ABB RobotStudio station: Compas_RRC_Course.rspag

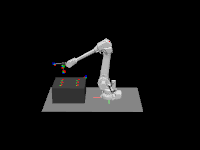
--- station ---
Station Compas_RRC_Course (saved by RobotStudio 20.4.9280.0)
Controller vIRB4600-40-255_RRC
  mechanical unit ROB_1: IRB4600_40_255_C_01, 6 joints, base frame (0, 0, 0) mm
Layout (positions relative to the parent item):
  - IRB4600_40_255_C_01 [mechanism] at (0, 0, 0) mm; joint values [0, -0.1281, 0.6287, 3.1416, 0.5005, 3.1416] (rad or m)
      links: Base, Link1, Link2, Link3, Link4, Link5, Link6
  - Table [part]
  - Ground [part]
  - Tool [graphiccomponentgroup] at (1368.26, 0, 1125.08) mm, rotated rx -13.36 ry 90 rz -13.36 deg
    - Tool X TubeTrace [smart component] at (0, 0, 0) mm
        properties: TraceObject=(none); ActiveTube=(none); Mechanism=IRB4600_40_255_C_01; Flange=Tool0; Parent=(none); Flange Offset=[0.26 0 0.06]; Tube Diameter=0.03; Color (RGB)=[255 255 255]; Color=-65536; Min Distance=0.001; Redraw Rate (ms)=10; NoOfBodies=210; Remove Geometry=true; Transient=false
        signals: DI Execute, DI NewTrace, DI Clear, DO TraceCreated
    - Tool Y TubeTrace [smart component] at (0, 0, 0) mm
        properties: TraceObject=(none); ActiveTube=(none); Mechanism=IRB4600_40_255_C_01; Flange=Tool0; Parent=(none); Flange Offset=[0 0.26 0.06]; Tube Diameter=0.03; Color (RGB)=[255 255 255]; Color=-16711872; Min Distance=0.001; Redraw Rate (ms)=10; NoOfBodies=208; Remove Geometry=true; Transient=false
        signals: DI Execute, DI NewTrace, DI Clear, DO TraceCreated
    - Tool Z TubeTrace [smart component] at (0, 0, 0) mm
        properties: TraceObject=(none); ActiveTube=(none); Mechanism=IRB4600_40_255_C_01; Flange=Tool0; Parent=(none); Flange Offset=[0 0 0.32]; Tube Diameter=0.03; Color (RGB)=[255 255 255]; Color=-16776961; Min Distance=0.001; Redraw Rate (ms)=10; NoOfBodies=210; Remove Geometry=true; Transient=false
        signals: DI Execute, DI NewTrace, DI Clear, DO TraceCreated
    - Tool X [part] at (0, 0, 0) mm
    - Tool Y [part] at (0, 0, 0) mm
    - Tool Z [part] at (0, 0, 0) mm
    - Base [part] at (1428.26, 0, 1185.08) mm, rotated rx 180 ry 0 rz -180 deg
Attachment: Tool is attached to IRB4600_40_255_C_01 / Link6
Station logic (signal -> signal, property => property):
  vIRB4600-40-255_RRC.doPrintTX -> Tool X TubeTrace.Execute
  vIRB4600-40-255_RRC.doPrintTY -> Tool Y TubeTrace.Execute
  vIRB4600-40-255_RRC.doPrintTZ -> Tool Z TubeTrace.Execute
Targets, tools, work objects and paths stored in the station and not in the controller backup, written as RAPID:
! task T_ROB1
MODULE X000_Tests
  PROC r_X000_Parh_Z()
    MoveJ pZStart,v200,fine,t_X000_Tool_Z\WObj:=ob_X000_Workplace;
    MoveL pZ1,v200,fine,t_X000_Tool_Z\WObj:=ob_X000_Workplace;
    MoveL pZ2,v200,fine,t_X000_Tool_Z\WObj:=ob_X000_Workplace;
  ENDPROC
  PROC r_X000_Parh_X()
    MoveJ pXStart,v200,fine,t_X000_Tool_X\WObj:=ob_X000_Workplace;
    MoveL pX1,v200,fine,t_X000_Tool_X\WObj:=ob_X000_Workplace;
    MoveL pX2,v200,fine,t_X000_Tool_X\WObj:=ob_X000_Workplace;
  ENDPROC
  PROC r_X000_Parh_Y()
    MoveJ pYStart,v200,fine,t_X000_Tool_Y\WObj:=ob_X000_Workplace;
    MoveL pY1,v200,fine,t_X000_Tool_Y\WObj:=ob_X000_Workplace;
    MoveL pY2,v200,fine,t_X000_Tool_Y\WObj:=ob_X000_Workplace;
  ENDPROC
ENDMODULE


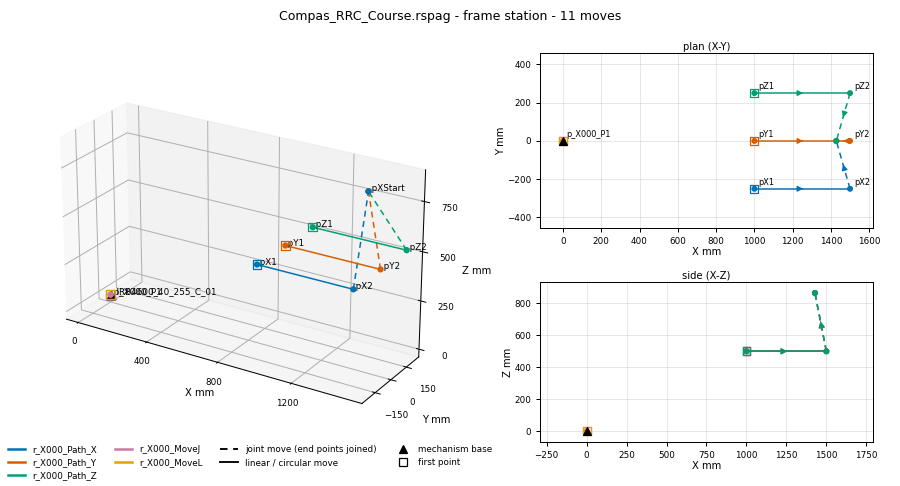
[picture p0: tool path of Compas_RRC_Course.rspag in frame station, 11 of 14 moves have a stored position in this frame; points joined in program order, loops and branches not executed]
--- Backups/vIRB4600-40-255_RRC/RAPID/TASK1/PROGMOD/X000_DataTask_1.mod ---
MODULE X000_DataTask_1
    !***********************************************************************************
    !
    ! ETH Zurich / NCCR Digital Fabrication
    ! HIB C51 / Stefano-Franscini-Platz 1
    ! CH-8093 Zürich
    !
    !***********************************************************************************
    !
    ! PROJECT     :  X000 Default
    !
    ! FUNCTION    :  Includ all Task Data's for Project
    !
    ! AUTHOR      :  Philippe Fleischmann
    !
    ! EMAIL       :  fleischmann@arch.ethz.ch
    !
    ! HISTORY     :  2019.12.04
    !
    ! Copyright   :  ETH Zürich (CH) 2019
    !
    !***********************************************************************************

    !************************************************
    ! Declaration :     bool
    !************************************************
    !

    !************************************************
    ! Declaration :     num
    !************************************************
    !

    !************************************************
    ! Declaration :     string
    !************************************************
    !

    !************************************************
    ! Declaration :     tooldata
    !************************************************
    !
    TASK PERS tooldata t_X000_Tool:=[TRUE,[[0,0,0],[1,0,0,0]],[1,[0,0,0],[1,0,0,0],0.1,0.1,0.1]];
    !
    TASK PERS tooldata t_X000_Tool_X:=[TRUE,[[260,0,60],[0.707106781,0,0.707106781,0]],[15,[0,0,60],[1,0,0,0],0.1,0.1,0.1]];
    TASK PERS tooldata t_X000_Tool_Y:=[TRUE,[[0,260,60],[0.707106781,-0.707106781,0,0]],[15,[0,0,60],[1,0,0,0],0.1,0.1,0.1]];
    TASK PERS tooldata t_X000_Tool_Z:=[TRUE,[[0,0,320],[1,0,0,0]],[15,[0,0,60],[1,0,0,0],0.1,0.1,0.1]];

    !************************************************
    ! Declaration :     wobjdata
    !************************************************
    !
    TASK PERS wobjdata ob_X000_Wobjdata:=[FALSE,TRUE,"",[[0,0,0],[1,0,0,0]],[[0,0,0],[1,0,0,0]]];
    !
    TASK PERS wobjdata ob_X000_Workplace:=[FALSE,TRUE,"",[[750,-500,500],[1,0,0,0]],[[0,0,0],[1,0,0,0]]];

    !************************************************
    ! Declaration :     jointtarget
    !************************************************
    !
    TASK PERS jointtarget jp_X000_Jointtarget:=[[0,0,0,0,0,0],[9E9,9E9,9E9,9E9,9E9,9E9]];
    !
    TASK PERS jointtarget jp_X000_Start:=[[1.2417E-18,-7.34132,36.0203,180,28.679,180],[9E+9,9E+9,9E+9,9E+9,9E+9,9E+9]];

    !************************************************
    ! Declaration :     robtarget
    !************************************************
    !
    TASK PERS robtarget p_X000_Robtarget:=[[0,0,0],[1,0,0,0],[0,0,0,0],[9E9,9E9,9E9,9E9,9E9,9E9]];

	CONST robtarget pXStart:=[[678.26315348,500,365.080626614],[0,0,1,0],[0,2,2,0],[9E+09,9E+09,9E+09,9E+09,9E+09,9E+09]];
	CONST robtarget pX1:=[[250.000037817,249.999985042,-0.000049799],[-0.000000001,0,1,-0.000000028],[-1,1,2,0],[9E+09,9E+09,9E+09,9E+09,9E+09,9E+09]];
	CONST robtarget pX2:=[[750.000017046,249.999996608,-0.000043508],[-0.000000001,-0.000000024,1,0],[-1,1,2,0],[9E+09,9E+09,9E+09,9E+09,9E+09,9E+09]];

    CONST robtarget pYStart:=[[678.26315348,500,365.080626614],[0,0,1,0],[0,-1,0,0],[9E+09,9E+09,9E+09,9E+09,9E+09,9E+09]];
	CONST robtarget pY1:=[[250.000037817,499.999985042,-0.000049799],[-0.000000001,0,1,-0.000000028],[0,-1,0,0],[9E+09,9E+09,9E+09,9E+09,9E+09,9E+09]];
	CONST robtarget pY2:=[[750.000017046,499.999996608,-0.000043508],[-0.000000001,-0.000000024,1,0],[0,-1,0,0],[9E+09,9E+09,9E+09,9E+09,9E+09,9E+09]];

    CONST robtarget pZStart:=[[678.26315348,500,365.080626614],[0,0,1,0],[0,0,0,0],[9E+09,9E+09,9E+09,9E+09,9E+09,9E+09]];
	CONST robtarget pZ1:=[[250.000037817,749.999985042,-0.000077799],[-0.000000001,0,1,-0.000000028],[0,-1,0,0],[9E+09,9E+09,9E+09,9E+09,9E+09,9E+09]];
	CONST robtarget pZ2:=[[750.000017046,749.999996608,-0.000071508],[-0.000000001,-0.000000024,1,0],[0,0,0,0],[9E+09,9E+09,9E+09,9E+09,9E+09,9E+09]];

    !************************************************
    ! Declaration :     speeddata
    !************************************************
    !
    TASK PERS speeddata v_X000_Speed:=[0,0,0,0];

ENDMODULE

--- Backups/vIRB4600-40-255_RRC/RAPID/TASK1/PROGMOD/X000_Demo.mod ---
MODULE X000_Demo
    !***********************************************************************************
    !
    ! ETH Zürich / Robotic Fabrication Lab
    ! HIB C 13 / Stefano-Franscini-Platz 1
    ! CH-8093 Zürich
    !
    !***********************************************************************************
    !
    ! PROJECT     :  X000_Default
    !
    ! FUNCTION    :  Demo
    !
    ! AUTHOR      :  Philippe Fleischmann
    !
    ! EMAIL       :  fleischmann@arch.ethz.ch
    !
    ! HISTORY     :  2021.01.14
    !
    ! Copyright   :  ETH Zürich (CH) 2021
    !
    !***********************************************************************************

    !************************************************
    ! Function    :     Demo x y and z path
    ! Programmer  :     Philippe Fleischmann
    ! Date        :     2021.01.14
    !***************** ETH Zürich *******************
    !
    PROC main()
        !
        ! Move to start point
        MoveAbsJ jp_X000_Start,v200,fine,tool0;
        !
        ! Test paths
        r_X000_Path_X;
        r_X000_Path_Y;
        r_X000_Path_Z;
        !
        ! Move to start point
        MoveAbsJ jp_X000_Start,v200,fine,tool0;
        !
        RETURN ;
    ERROR
        ! Placeholder for Error Code...
    ENDPROC

    !************************************************
    ! Function    :     Print Path red
    ! Programmer  :     Philippe Fleischmann
    ! Date        :     2021.01.14
    !***************** ETH Zürich *******************
    !
    PROC r_X000_Path_X()
        !
        ! Move to print start
        MoveJ pX1,v200,fine,t_X000_Tool_X\WObj:=ob_X000_Workplace;
        !
        ! Start print
        SetDO doPrintTX,1;
        !
        ! Print
        MoveL pX2,v200,fine,t_X000_Tool_X\WObj:=ob_X000_Workplace;
        !
        ! Stop pring
        SetDO doPrintTX,0;
        !
        ! Move back to start point
        MoveJ pXStart,v200,fine,t_X000_Tool_X\WObj:=ob_X000_Workplace;
        !
        RETURN ;
    ERROR
        ! Placeholder for Error Code...
    ENDPROC

    !************************************************
    ! Function    :     Print Path green
    ! Programmer  :     Philippe Fleischmann
    ! Date        :     2021.01.14
    !***************** ETH Zürich *******************
    !
    PROC r_X000_Path_Y()
        !
        ! Move to print start
        MoveJ pY1,v200,fine,t_X000_Tool_Y\WObj:=ob_X000_Workplace;
        !
        ! Start print
        SetDO doPrintTY,1;
        !
        ! Print
        MoveL pY2,v200,fine,t_X000_Tool_Y\WObj:=ob_X000_Workplace;
        !
        ! Stop pring
        SetDO doPrintTY,0;
        !
        ! Move back to start point
        MoveJ pYStart,v200,fine,t_X000_Tool_Y\WObj:=ob_X000_Workplace;
        !
        RETURN ;
    ERROR
        ! Placeholder for Error Code...
    ENDPROC

    !************************************************
    ! Function    :     Print Path blue
    ! Programmer  :     Philippe Fleischmann
    ! Date        :     2021.01.14
    !***************** ETH Zürich *******************
    !
    PROC r_X000_Path_Z()
        !
        ! Move to print start
        MoveJ pZ1,v200,fine,t_X000_Tool_Z\WObj:=ob_X000_Workplace;
        !
        ! Start print
        SetDO doPrintTZ,1;
        !
        ! Print
        MoveL pZ2,v200,fine,t_X000_Tool_Z\WObj:=ob_X000_Workplace;
        !
        ! Stop pring
        SetDO doPrintTZ,0;
        !
        ! Move back to start point
        MoveJ pZStart,v200,fine,t_X000_Tool_Z\WObj:=ob_X000_Workplace;
        !
        RETURN ;
    ERROR
        ! Placeholder for Error Code...
    ENDPROC

ENDMODULE

--- Backups/vIRB4600-40-255_RRC/RAPID/TASK1/PROGMOD/X000_Motion.mod ---
MODULE X000_Motion
    !***********************************************************************************
    !
    ! ETH Zürich / Robotic Fabrication Lab
    ! HIB C 13 / Stefano-Franscini-Platz 1
    ! CH-8093 Zürich
    !
    !***********************************************************************************
    !
    ! PROJECT     :  X000_Default
    !
    ! FUNCTION    :  Motion Types
    !
    ! AUTHOR      :  Philippe Fleischmann
    !
    ! EMAIL       :  fleischmann@arch.ethz.ch
    !
    ! HISTORY     :  2020.01.09
    !
    ! Copyright   :  ETH Zürich (CH) 2017
    !
    !***********************************************************************************

    !************************************************
    ! Declaration :     jointtarget
    !************************************************
    !
    TASK PERS jointtarget jp_X000_P1:=[[0,0,0,0,0,0],[9E9,9E9,9E9,9E9,9E9,9E9]];

    !************************************************
    ! Declaration :     robtarget
    !************************************************
    !
    TASK PERS robtarget p_X000_P1:=[[0,0,0],[1,0,0,0],[0,0,0,0],[9E9,9E9,9E9,9E9,9E9,9E9]];

    !************************************************
    ! Function    :     Move absolute Joint
    ! Programmer  :     Philippe Fleischmann
    ! Date        :     2020.01.07
    !***************** ETH Zürich *******************
    !
    PROC r_X000_MoveAbsJ()
        !
        ! MoveAbsJ
        MoveAbsJ jp_X000_P1,v100,fine,tool0;
        !
        RETURN ;
    ERROR
        ! Placeholder for Error Code...
    ENDPROC

    !************************************************
    ! Function    :     Move Joint
    ! Programmer  :     Philippe Fleischmann
    ! Date        :     2020.01.07
    !***************** ETH Zürich *******************
    !
    PROC r_X000_MoveJ()
        !
        ! MoveJ
        MoveJ p_X000_P1,v100,fine,tool0\WObj:=wobj0;
        !
        RETURN ;
    ERROR
        ! Placeholder for Error Code...
    ENDPROC

    !************************************************
    ! Function    :     Move Linear
    ! Programmer  :     Philippe Fleischmann
    ! Date        :     2020.01.07
    !***************** ETH Zürich *******************
    !
    PROC r_X000_MoveL()
        !
        ! MoveL
        MoveL p_X000_P1,v100,fine,tool0\WObj:=wobj0;
        !
        RETURN ;
    ERROR
        ! Placeholder for Error Code...
    ENDPROC

ENDMODULE

--- Backups/vIRB4600-40-255_RRC/SYSPAR/EIO.cfg ---
EIO:CFG_1.0:6:1::
#
INDUSTRIAL_NETWORK:

      -Name "PROFINET" -Connection "PROFINET Network"\
      -Label "PROFINET Controller/Device Network" -StationName ""
#
EIO_CROSS:

      -Name "FP1" -Res "diMaFP1" -Act1 "doMaFP1"

      -Name "FP2" -Res "diMaFP2" -Act1 "doMaFP2"

      -Name "FP3" -Res "diMaFP3" -Act1 "doMaFP3"

      -Name "FP4" -Res "diMaFP4" -Act1 "doMaFP4"
#
EIO_ACCESS:

      -Name "RFL_Safe" -Rapid
#
PROFINET_DRIVER:

      -Name "PROFINET_COMMON_DATA"
#
PROFINET_INTERNAL_DEVICE:

      -Name "PN_Internal_Device" -VendorName "ABB Robotics"\
      -ProductName "PROFINET Internal Device"
#
EIO_SIGNAL:

      -Name "diMaFP1" -SignalType "DI"\
      -Label "Virtual - Master FlexPendant Taste 1" -DeviceMap "0" -Access "All"

      -Name "diMaFP2" -SignalType "DI"\
      -Label "Virtual - Master FlexPendant Taste 2" -DeviceMap "1" -Access "All"

      -Name "diMaFP3" -SignalType "DI"\
      -Label "Virtual - Master FlexPendant Taste 3" -DeviceMap "2" -Access "All"

      -Name "diMaFP4" -SignalType "DI"\
      -Label "Virtual - Master FlexPendant Taste 4" -DeviceMap "3" -Access "All"

      -Name "diMaActSpLi" -SignalType "DI"\
      -Label "Virtual - Master Activate Speed Limit" -DeviceMap "4"\
      -Access "All"

      -Name "diMaReset" -SignalType "DI" -Label "Virtual - Master Reset"\
      -DeviceMap "5" -Access "All"

      -Name "diMaRes7" -SignalType "DI" -Label "Virtual - Master Reserve 7"\
      -DeviceMap "6" -Access "All"

      -Name "diMaRes8" -SignalType "DI" -Label "Virtual - Master Reserve 8"\
      -DeviceMap "7" -Access "All"

      -Name "doMaFP1" -SignalType "DO"\
      -Label "Virtual - Master FlexPendant Taste 1" -DeviceMap "0" -Access "All"

      -Name "doMaFP2" -SignalType "DO"\
      -Label "Virtual - Master FlexPendant Taste 2" -DeviceMap "1" -Access "All"

      -Name "doMaFP3" -SignalType "DO"\
      -Label "Virtual - Master FlexPendant Taste 3" -DeviceMap "2" -Access "All"

      -Name "doMaFP4" -SignalType "DO"\
      -Label "Virtual - Master FlexPendant Taste 4" -DeviceMap "3" -Access "All"

      -Name "doMaSpLiAct" -SignalType "DO"\
      -Label "Virtual - Master Speed Limit Activ" -DeviceMap "4" -Access "All"

      -Name "doMaReset" -SignalType "DO" -Label "Virtual - Master Reset"\
      -DeviceMap "5" -Access "All"

      -Name "doMaRes7" -SignalType "DO" -Label "Virtual - Master Reserve 7"\
      -DeviceMap "6" -Access "All"

      -Name "doMaRes8" -SignalType "DO" -Label "Virtual - Master Reserve 8"\
      -DeviceMap "7" -Access "All"

      -Name "doPrintTX" -SignalType "DO"

      -Name "doPrintTY" -SignalType "DO"

      -Name "doPrintTZ" -SignalType "DO"
